VAR_GLOBAL
	timer0: TON;
	timer1: TON;
	curTimer: INT := 0;
END_VAR

(* stored: Version 1.1.0.1, ProductVersion 3.1.4022.18
   GVL TIMERS: Id {15d04d52-1246-4e2f-a09e-65bcbb826634} *)
